Fanuc TP program (LS listing): ROUTER.LS

/PROG  ROUTER	  Macro
/ATTR
OWNER		= MNEDITOR;
COMMENT		= "Pounce Router";
PROG_SIZE	= 6945;
CREATE		= DATE 22-07-01  TIME 07:23:44;
MODIFIED	= DATE 29-06-14  TIME 05:04:00;
FILE_NAME	= ;
VERSION		= 0;
LINE_COUNT	= 366;
MEMORY_SIZE	= 7953;
PROTECT		= READ_WRITE;
TCD:  STACK_SIZE	= 1200,
      TASK_PRIORITY	= 50,
      TIME_SLICE	= 0,
      BUSY_LAMP_OFF	= 0,
      ABORT_REQUEST	= 0,
      PAUSE_REQUEST	= 0;
DEFAULT_GROUP	= 1,*,*,*,*;
CONTROL_CODE	= 00000000 00000000;
/APPL
/APPL

LINE_TRACK;
  LINE_TRACK_SCHEDULE_NUMBER      : 0;
  LINE_TRACK_BOUNDARY_NUMBER      : 0;
  CONTINUE_TRACK_AT_PROG_END      : FALSE;

/MN
   1:  !******************************* ;
   2:  !COMPANY ;
   3:  !PROJECT 0000000 ;
   4:  !CUSTOMER ;
   5:  ! ;
   6:  !Date: February 10, 2020 ;
   7:  ! ;
   8:  !Router for paths between ;
   9:  !pounce positions ;
  10:  ! ;
  11:  !******************************* ;
  12:  LBL[1:Begin] ;
  13:   ;
  14:  !Set Move Defaults ;
  15:  R[11:Router Speed]=40    ;
  16:  R[12:Router CNT Value]=70    ;
  17:  R[100:Max Recov Dist]=25    ;
  18:  R[101:Number Perches]=7    ;
  19:  R[102:First Perch PR#]=1    ;
  20:  R[104:Curr Perch PR#]=0    ;
  21:   ;
  22:  UFRAME_NUM=1 ;
  23:  UTOOL_NUM=1 ;
  24:   ;
  25:  !Set destination reg ;
  26:  R[103:Dest Perch PR#]=AR[1]    ;
  27:   ;
  28:  LBL[2:Check] ;
  29:  !Check current position ;
  30:  IF R[104:Curr Perch PR#]=0,JMP LBL[3] ;
  31:   ;
  32:  R[111]=R[102:First Perch PR#]+R[101:Number Perches]-1    ;
  33:   ;
  34:  !Range check curr ;
  35:  IF R[104:Curr Perch PR#]<R[102:First Perch PR#] OR R[104:Curr Perch PR#]>R[111],JMP LBL[5000] ;
  36:   ;
  37:  !Range check dest ;
  38:  IF R[103:Dest Perch PR#]<R[102:First Perch PR#] OR R[103:Dest Perch PR#]>R[111],JMP LBL[5100] ;
  39:   ;
  40:  !Robot must be at current perch ;
  41:  IF SO[7:TP enabled]=ON,JMP LBL[3] ;
  42:  IF R[104:Curr Perch PR#]=0,JMP LBL[3] ;
  43:  JMP LBL[4] ;
  44:   ;
  45:  LBL[3:Find Posn] ;
  46:  CALL RECOVERY    ;
  47:  CALL GET_POS    ;
  48:  IF R[104:Curr Perch PR#]<>0,JMP LBL[4] ;
  49:  DO[58:TP Input Required]=ON ;
  50:  CALL GO_PERCH    ;
  51:  DO[58:TP Input Required]=OFF ;
  52:  JMP LBL[2] ;
  53:   ;
  54:   ;
  55:  !-------------------------------- ;
  56:  LBL[4:Select From PosR] ;
  57:  !-------------------------------- ;
  58:  SELECT R[104:Curr Perch PR#]=1,JMP LBL[100] ;
  59:         =2,JMP LBL[200] ;
  60:         =3,JMP LBL[300] ;
  61:         =4,JMP LBL[400] ;
  62:         =5,JMP LBL[500] ;
  63:         =6,JMP LBL[600] ;
  64:         =7,JMP LBL[700] ;
  65:         ELSE,JMP LBL[5000] ;
  66:   ;
  67:   ;
  68:  !-------------------------------- ;
  69:  LBL[100:From PR1(Home)] ;
  70:  !-------------------------------- ;
  71:  SELECT R[103:Dest Perch PR#]=1,JMP LBL[101] ;
  72:         =2,JMP LBL[102] ;
  73:         =3,JMP LBL[103] ;
  74:         =4,JMP LBL[104] ;
  75:         =5,JMP LBL[105] ;
  76:         =6,JMP LBL[106] ;
  77:         =7,JMP LBL[107] ;
  78:         ELSE,JMP LBL[5000] ;
  79:   ;
  80:  LBL[101:To PR1(Home)] ;
  81:  JMP LBL[4950] ;
  82:   ;
  83:  LBL[102:To PR2(Maint)] ;
  84:J PR[2:Maint Perch] 25% CNT80    ;
  85:  JMP LBL[4950] ;
  86:   ;
  87:  LBL[103:To PR3 Outfd] ;
  88:  JMP LBL[4950] ;
  89:   ;
  90:  LBL[104:To PR4 Grd] ;
  91:J PR[4:Grinder Perch] 15% CNT80    ;
  92:  JMP LBL[4950] ;
  93:   ;
  94:  LBL[105:To PR5 Hanoff] ;
  95:  JMP LBL[4950] ;
  96:   ;
  97:  LBL[106:To PR6 Vis] ;
  98:  JMP LBL[4950] ;
  99:   ;
 100:  LBL[107:To PR7(Audit)] ;
 101:J PR[7:Audit] 10% FINE    ;
 102:  JMP LBL[4950] ;
 103:   ;
 104:  !-------------------------------- ;
 105:  LBL[200:From PR2(Maint)] ;
 106:  !-------------------------------- ;
 107:  SELECT R[103:Dest Perch PR#]=1,JMP LBL[201] ;
 108:         =2,JMP LBL[202] ;
 109:         =3,JMP LBL[203] ;
 110:         =4,JMP LBL[204] ;
 111:         =5,JMP LBL[205] ;
 112:         =6,JMP LBL[206] ;
 113:         =7,JMP LBL[207] ;
 114:         ELSE,JMP LBL[5000] ;
 115:   ;
 116:  LBL[201:To PR1(Home)] ;
 117:J PR[1:Robot Home] 25% CNT25    ;
 118:  JMP LBL[4950] ;
 119:   ;
 120:  LBL[202:To PR2(Maint)] ;
 121:  JMP LBL[4950] ;
 122:   ;
 123:  LBL[203:To PR3(Outfd)] ;
 124:  JMP LBL[4950] ;
 125:   ;
 126:  LBL[204:To PR4(Grid)] ;
 127:J PR[4:Grinder Perch] 15% CNT80    ;
 128:  JMP LBL[4950] ;
 129:   ;
 130:  LBL[205:To PR5(Handoff)] ;
 131:  JMP LBL[4950] ;
 132:   ;
 133:  LBL[206:To PR6(Vision)] ;
 134:J PR[1:Robot Home] 40% CNT80    ;
 135:  JMP LBL[4950] ;
 136:   ;
 137:  LBL[207:To PR7(Audit)] ;
 138:J PR[1:Robot Home] 40% CNT80    ;
 139:J PR[7:Audit] 10% FINE    ;
 140:  JMP LBL[4950] ;
 141:   ;
 142:  !-------------------------------- ;
 143:  LBL[300:From PR3(Outfee)] ;
 144:  !-------------------------------- ;
 145:  SELECT R[103:Dest Perch PR#]=1,JMP LBL[301] ;
 146:         =2,JMP LBL[302] ;
 147:         =3,JMP LBL[303] ;
 148:         =4,JMP LBL[304] ;
 149:         =5,JMP LBL[305] ;
 150:         =6,JMP LBL[306] ;
 151:         =7,JMP LBL[307] ;
 152:         ELSE,JMP LBL[5000] ;
 153:   ;
 154:  LBL[301:To PR1(Home)] ;
 155:  JMP LBL[4950] ;
 156:   ;
 157:  LBL[302:To PR2(Maint)] ;
 158:  JMP LBL[4950] ;
 159:   ;
 160:  LBL[303:To PR3(OutFd)] ;
 161:  JMP LBL[4950] ;
 162:   ;
 163:  LBL[304:To PR4(Grd)] ;
 164:J PR[1:Robot Home] 15% CNT80    ;
 165:J PR[4:Grinder Perch] 15% CNT80    ;
 166:  JMP LBL[4950] ;
 167:   ;
 168:  LBL[305:To PR5(Handoff)] ;
 169:  JMP LBL[4950] ;
 170:   ;
 171:  LBL[306:To PR6(Vision)] ;
 172:J PR[1:Robot Home] 10% CNT80    ;
 173:  JMP LBL[4950] ;
 174:   ;
 175:  LBL[307:To PR7(Audit)] ;
 176:J PR[7:Audit] 10% CNT80    ;
 177:  JMP LBL[4950] ;
 178:   ;
 179:  !-------------------------------- ;
 180:  LBL[400:From PR4(Grd)] ;
 181:  !-------------------------------- ;
 182:  SELECT R[103:Dest Perch PR#]=1,JMP LBL[401] ;
 183:         =2,JMP LBL[402] ;
 184:         =3,JMP LBL[403] ;
 185:         =4,JMP LBL[404] ;
 186:         =5,JMP LBL[405] ;
 187:         =6,JMP LBL[406] ;
 188:         =7,JMP LBL[407] ;
 189:         ELSE,JMP LBL[5000] ;
 190:   ;
 191:  LBL[401:To PR1(Home)] ;
 192:J PR[1:Robot Home] 25% CNT25    ;
 193:  JMP LBL[4950] ;
 194:   ;
 195:  LBL[402:To PR2(Maint)] ;
 196:  JMP LBL[4950] ;
 197:   ;
 198:  LBL[403:To PR3(OutFd)] ;
 199:J PR[1:Robot Home] 30% CNT80    ;
 200:  JMP LBL[4950] ;
 201:   ;
 202:  LBL[404:To PR4(Grd)] ;
 203:  JMP LBL[4950] ;
 204:   ;
 205:  LBL[405:To PR5(Handoff) ] ;
 206:  JMP LBL[4950] ;
 207:   ;
 208:  LBL[406:To PR6(Vision)] ;
 209:J PR[1:Robot Home] 25% CNT80    ;
 210:  JMP LBL[4950] ;
 211:   ;
 212:  LBL[407:To PR7(Audit)] ;
 213:J PR[1:Robot Home] 40% CNT80    ;
 214:J PR[7:Audit] 10% FINE    ;
 215:  JMP LBL[4950] ;
 216:   ;
 217:  !-------------------------------- ;
 218:  LBL[500:From PR5(Handof)] ;
 219:  !-------------------------------- ;
 220:  SELECT R[103:Dest Perch PR#]=1,JMP LBL[501] ;
 221:         =2,JMP LBL[502] ;
 222:         =3,JMP LBL[503] ;
 223:         =4,JMP LBL[504] ;
 224:         =5,JMP LBL[505] ;
 225:         =6,JMP LBL[506] ;
 226:         =7,JMP LBL[507] ;
 227:         ELSE,JMP LBL[5000] ;
 228:   ;
 229:  LBL[501:To PR1(Home)] ;
 230:  JMP LBL[4950] ;
 231:   ;
 232:  LBL[502:To PR2(Maint)] ;
 233:  JMP LBL[4950] ;
 234:   ;
 235:  LBL[503:To PR3(OutFd)] ;
 236:  JMP LBL[4950] ;
 237:   ;
 238:  LBL[504:To PR4(Grd)] ;
 239:J PR[4:Grinder Perch] 15% CNT80    ;
 240:  JMP LBL[4950] ;
 241:   ;
 242:  LBL[505:To PR5(Handoff)] ;
 243:  JMP LBL[4950] ;
 244:   ;
 245:  LBL[506:To PR6(Vision)] ;
 246:  JMP LBL[4950] ;
 247:   ;
 248:  LBL[507:To PR7(Audit)] ;
 249:J PR[1:Robot Home] 40% CNT80    ;
 250:J PR[7:Audit] 10% FINE    ;
 251:  JMP LBL[4950] ;
 252:   ;
 253:  !-------------------------------- ;
 254:  LBL[600:From PR6(Vision)] ;
 255:  !-------------------------------- ;
 256:  SELECT R[103:Dest Perch PR#]=1,JMP LBL[601] ;
 257:         =2,JMP LBL[602] ;
 258:         =3,JMP LBL[603] ;
 259:         =4,JMP LBL[604] ;
 260:         =5,JMP LBL[605] ;
 261:         =6,JMP LBL[606] ;
 262:         =7,JMP LBL[607] ;
 263:         ELSE,JMP LBL[5000] ;
 264:   ;
 265:  LBL[601:To PR1(Home)] ;
 266:  JMP LBL[4950] ;
 267:   ;
 268:  LBL[602:To PR2(Maint)] ;
 269:J PR[1:Robot Home] 10% FINE    ;
 270:  JMP LBL[4950] ;
 271:   ;
 272:  LBL[603:To PR3(OutFd)] ;
 273:J PR[1:Robot Home] 20% CNT25    ;
 274:  JMP LBL[4950] ;
 275:   ;
 276:  LBL[604:To PR4(Grd)] ;
 277:J PR[1:Robot Home] 50% CNT80    ;
 278:J PR[4:Grinder Perch] 15% CNT80    ;
 279:  JMP LBL[4950] ;
 280:   ;
 281:  LBL[605:To PR5(Handoff)] ;
 282:  JMP LBL[4950] ;
 283:   ;
 284:  LBL[606:To PR6(Vision)] ;
 285:  JMP LBL[4950] ;
 286:   ;
 287:  LBL[607:To PR7(Audit) ] ;
 288:J PR[1:Robot Home] 40% CNT80    ;
 289:J PR[7:Audit] 10% FINE    ;
 290:  JMP LBL[4950] ;
 291:   ;
 292:  !-------------------------------- ;
 293:  LBL[700:From PR7(Audit)] ;
 294:  !-------------------------------- ;
 295:  SELECT R[103:Dest Perch PR#]=1,JMP LBL[701] ;
 296:         =2,JMP LBL[702] ;
 297:         =3,JMP LBL[703] ;
 298:         =4,JMP LBL[704] ;
 299:         =5,JMP LBL[705] ;
 300:         =6,JMP LBL[706] ;
 301:         =7,JMP LBL[707] ;
 302:         ELSE,JMP LBL[5000] ;
 303:   ;
 304:  LBL[701:To PR1(Home)] ;
 305:J PR[1:Robot Home] 25% CNT75    ;
 306:  JMP LBL[4950] ;
 307:   ;
 308:  LBL[702:To PR2(Maint)] ;
 309:J PR[1:Robot Home] 25% CNT50    ;
 310:J PR[2:Maint Perch] 25% CNT25    ;
 311:  JMP LBL[4950] ;
 312:   ;
 313:  LBL[703:To PR3(OutFd)] ;
 314:J PR[3:Outfeed Perch] 10% CNT10    ;
 315:  JMP LBL[4950] ;
 316:   ;
 317:  LBL[704:To PR4(Grd)] ;
 318:J PR[4:Grinder Perch] 15% CNT80    ;
 319:  JMP LBL[4950] ;
 320:   ;
 321:  LBL[705:To PR5(Handoff)] ;
 322:  JMP LBL[4950] ;
 323:   ;
 324:  LBL[706:To PR6(Vision)] ;
 325:J PR[1:Robot Home] 25% CNT50    ;
 326:  JMP LBL[4950] ;
 327:   ;
 328:  LBL[707:To PR7(Audit)] ;
 329:  JMP LBL[4950] ;
 330:   ;
 331:  !-------------------------------- ;
 332:  LBL[4950:Joint To Dest] ;
 333:  !-------------------------------- ;
 334:J PR[R[103]] R[10:Audit Router Spd]% CNT R[12:Router CNT Value]    ;
 335:  R[104:Curr Perch PR#]=R[103:Dest Perch PR#]    ;
 336:   ;
 337:  CALL ALL_CLR    ;
 338:  END ;
 339:   ;
 340:  !-------------------------------- ;
 341:  LBL[4960:Linear To Dest] ;
 342:  !-------------------------------- ;
 343:L PR[R[103]] 2000mm/sec CNT R[12:Router CNT Value]    ;
 344:  R[104:Curr Perch PR#]=R[103:Dest Perch PR#]    ;
 345:   ;
 346:  CALL ALL_CLR    ;
 347:  END ;
 348:   ;
 349:   ;
 350:  !******************************* ;
 351:  !FAULTS ;
 352:  !******************************* ;
 353:  LBL[5000] ;
 354:  !Router R[103] Out of Range ;
 355:  UALM[51] ;
 356:  ABORT ;
 357:   ;
 358:  LBL[5100] ;
 359:  !Router R[104] Out of Range ;
 360:  UALM[52] ;
 361:  ABORT ;
 362:   ;
 363:  LBL[5200] ;
 364:  !Router Unplanned Path ;
 365:  UALM[52] ;
 366:  ABORT ;
/POS
/END
